// TIA Portal V20 export
TYPE "UDT_Service_ParameterDefinition"
   STRUCT
      indexMTP : Int;   // Index of parameter / MTP Index of parameter
      indexIO : Int;   // Index of parameter / IO Index of parameter
      "type" : Int;   // Type of parameter
      controlModule : Byte := 16#FF;   // Number of control module used with parameter
   END_STRUCT;
END_TYPE
